(* IEC 61131-3 sources: POMIRTS_lab3/AS/Library/AsUPS, 2 files *)

(* ---- AsUPS.fun ---- *)
(********************************************************************
 * COPYRIGHT -- Bernecker + Rainer
 ********************************************************************
 * Library: AsUPS
 * File: AsUPS.fun
 * Author: B+R
 ********************************************************************
 * Functions and function blocks of library AsUPS
 ********************************************************************)

FUNCTION_BLOCK ups_comm					(*transfers additional parameters and commands to the UPS*)
	VAR_INPUT
		enable	:BOOL;					(*enables execution*)
		user_command	:STRING[128];	(*string which should be transferred to the UPS*)
	END_VAR
	VAR_OUTPUT
		status	:UINT;					(*execution status: ERR_OK, ERR_FUB_ENABLE_FALSE, 0xXXXX = see help*)
		ups_answer	:STRING[128];		(*response from the UPS*)
	END_VAR
END_FUNCTION_BLOCK

FUNCTION_BLOCK ups_init					(*initializes the connection and transfer of UPS parameters*)
	VAR_INPUT
		enable	:BOOL;					(*enables execution*)
		device	:UDINT;					(*device name given as a pointer, which clearly describes the interface used*)
		mode	:UDINT;					(*string which configures the interface to be used, given as a pointer*)
		ShutDownTime	:DINT;			(*time from the detection of the UPS shutdown message to the time it takes automation runtime to shut down*)
		ShutDownMode	:USINT;			(*parameter for shutdown mode: 0 no shutdown, 17 shutdown with warm restart mode, ..*)
		ShutDownDCD	:USINT;				(*shutdown condition for the DCD signal*)
		TWL	:STRING[10];				(*parameter for TWL example*)
		LCS	:STRING[10];				(*parameter for LCS*)
		SDT	:STRING[10];				(*parameter for SDT*)
		POT	:STRING[10];				(*parameter for POT*)
	END_VAR
	VAR_OUTPUT
		status	:UINT;					(*execution status: ERR_OK, ERR_FUB_ENABLE_FALSE, 0xXXXX = see help*)
		UPS_OS	:STRING[128];			(*UPS operating system version*)
	END_VAR
END_FUNCTION_BLOCK

FUNCTION_BLOCK ups_getcomstate			(*monitors handshake transmissions and shutdowns for automation runtime*)
	VAR_INPUT
		enable	:BOOL;					(*enables execution*)
	END_VAR
	VAR_OUTPUT
		status	:UINT;					(*execution status: ERR_OK, ERR_FUB_ENABLE_FALSE, 0xXXXX = see help*)
		DCD	:BOOL;						(*DCD signal state*)
		CTS	:BOOL;						(*CTS signal state*)
		ShutDownTime	:REAL;			(*delay time until automation runtime shutdown*)
	END_VAR
	VAR
		DCD_old	:BOOL;					(*internal variable*)
		CTS_old	:BOOL;					(*internal variable*)
	END_VAR
END_FUNCTION_BLOCK

FUNCTION ups_ar_shutdown : UINT			(*restarts or shuts down automation runtime*)
	VAR_INPUT
		enable	:BOOL;					(*enables execution*)
		ShutDownMode	:USINT;			(*shutdown mode: 0 no shutdown, 01 restart with warm restart mode, ..*)
	END_VAR
END_FUNCTION

FUNCTION ups_deinit : UINT				(*closes all internal connections and releases the interface*)
	VAR_INPUT
		enable	:BOOL;					(*enables execution*)
	END_VAR
END_FUNCTION

(* ---- AsUPS.var ---- *)
(********************************************************************
 * COPYRIGHT -- Bernecker + Rainer
 ********************************************************************
 * Library: AsUPS
 * File: AsUPS.var
 * Author: B+R
 ********************************************************************
 * Local variables of library AsUPS
 ********************************************************************)

VAR CONSTANT
	err_STARTSHUTDOWN	: UINT	:= 28260;			(*shutdown message from the UPS was detected*)
	SHUTDOWNWARMSTART	: USINT	:= 17;				(*WARMSTART (no restart, only shutdown, waits for "power off", in connection with UPS)*)
	SHUTDOWNCOLDSTART	: USINT	:= 18;				(*COLDSTART (no restart, only shutdown, waits for "power off", in connection with UPS)*)
	RESTARTWARMSTART	: USINT	:= 1;				(*WARMSTART (with restart)*)
	RESTARTCOLDSTART	: USINT	:= 2;				(*COLDSTART (with restart)*)
	ERR_LOWCYCLETIME	: UINT	:= 28259;			(*functions are called in a task class with a cycle time less than 10 ms*)
	INVALID_STRING	: STRING[20]	:= 'invalid';	(*'invalid'*)
	ERR_NOTDEFINED	: UINT	:= 28257;				(*unknown command or mode given*)
	ERR_NOSHUTDOWN	: UINT	:= 28258;				(*0x11 or 0x12 was not given as a ShutDownMode / Automation Runtime was not shutdown*)
	ERR_UPSANSWER	: UINT	:= 28252;				(*error response from the UPS*)
	ERR_SHUTDOWN	: UINT	:= 28251;				(*automation runtime is shutdown*)
	ERR_PROGRAMM	: UINT	:= 28253;				(*internal program error*)
	ERR_RESTART	: UINT	:= 28250;					(*automation runtime is restarted*)
	ERR_NOTINIT	: UINT	:= 28256;					(*ups_init not called*)
	ERR_NOINPUT	: UINT	:= 60;						(*no message received*)
	ERR_ENABLE0	: UINT	:= 65534;					(*FBK input enable = FALSE*)
	UPS_STRING	: STRING[20]	:= 'USV';			(*'USV'*)
	UPG_STRING	: STRING[20]	:= 'UPG';			(*'UPG'*)
	ERR_STRING	: STRING[20]	:= 'err';			(*'err'*)
	err_UPSOK	: UINT	:= 28261;					(*UPS did not receive an error and is in normal mode (power supply ok)*)
	OK_STRING	: STRING[20]	:= 'OK!';			(*'OK!'*)
	ERR_READY	: UINT	:= 0;						(*FBK executed correctly with no errors*)
	ERR_BUSY	: UINT	:= 65535;					(*FBK not yet complete - call FBK again*)
	ERR_DCD	: UINT	:= 28254;						(*change in DCD detected*)
	ERR_CTS	: UINT	:= 28255;						(*change in CTS detected*)
END_VAR
